TYPE SM_HMI_cfg :
STRUCT
  Name : STRING(40);
  HomePerm : ST_PermIntlk_HMI;
  StartPerm : ST_PermIntlk_HMI;
  ProceedPerm : ST_PermIntlk_HMI;
  AutoIntlk : ST_PermIntlk_HMI;
END_STRUCT
END_TYPE

(* stored: Version 1.1.0.1, ProductVersion 3.1.4024.13
   DUT SM_HMI_cfg: Id {4edb47ef-88d7-4424-b458-d70f5be9e1ea} *)
